INTERFACE iTracePublisher EXTENDS iBase

METHOD Subscribe
VAR_INPUT
	Logger : iTraceLogger;
END_VAR
END_METHOD

METHOD Unsubscribe
VAR_INPUT
	Logger : iTraceLogger;
END_VAR
END_METHOD

END_INTERFACE

(* stored: Version 1.1.0.1, ProductVersion 3.1.4026.18
   Itf iTracePublisher: Id {d510580b-a344-4b7a-a506-8b6d5e862184}
   Method Subscribe: Id {756f524e-6487-44ac-b3e2-883bf3b1f74c}
   Method Unsubscribe: Id {0a67286e-4060-4ba3-8a49-c0472d76b433} *)
